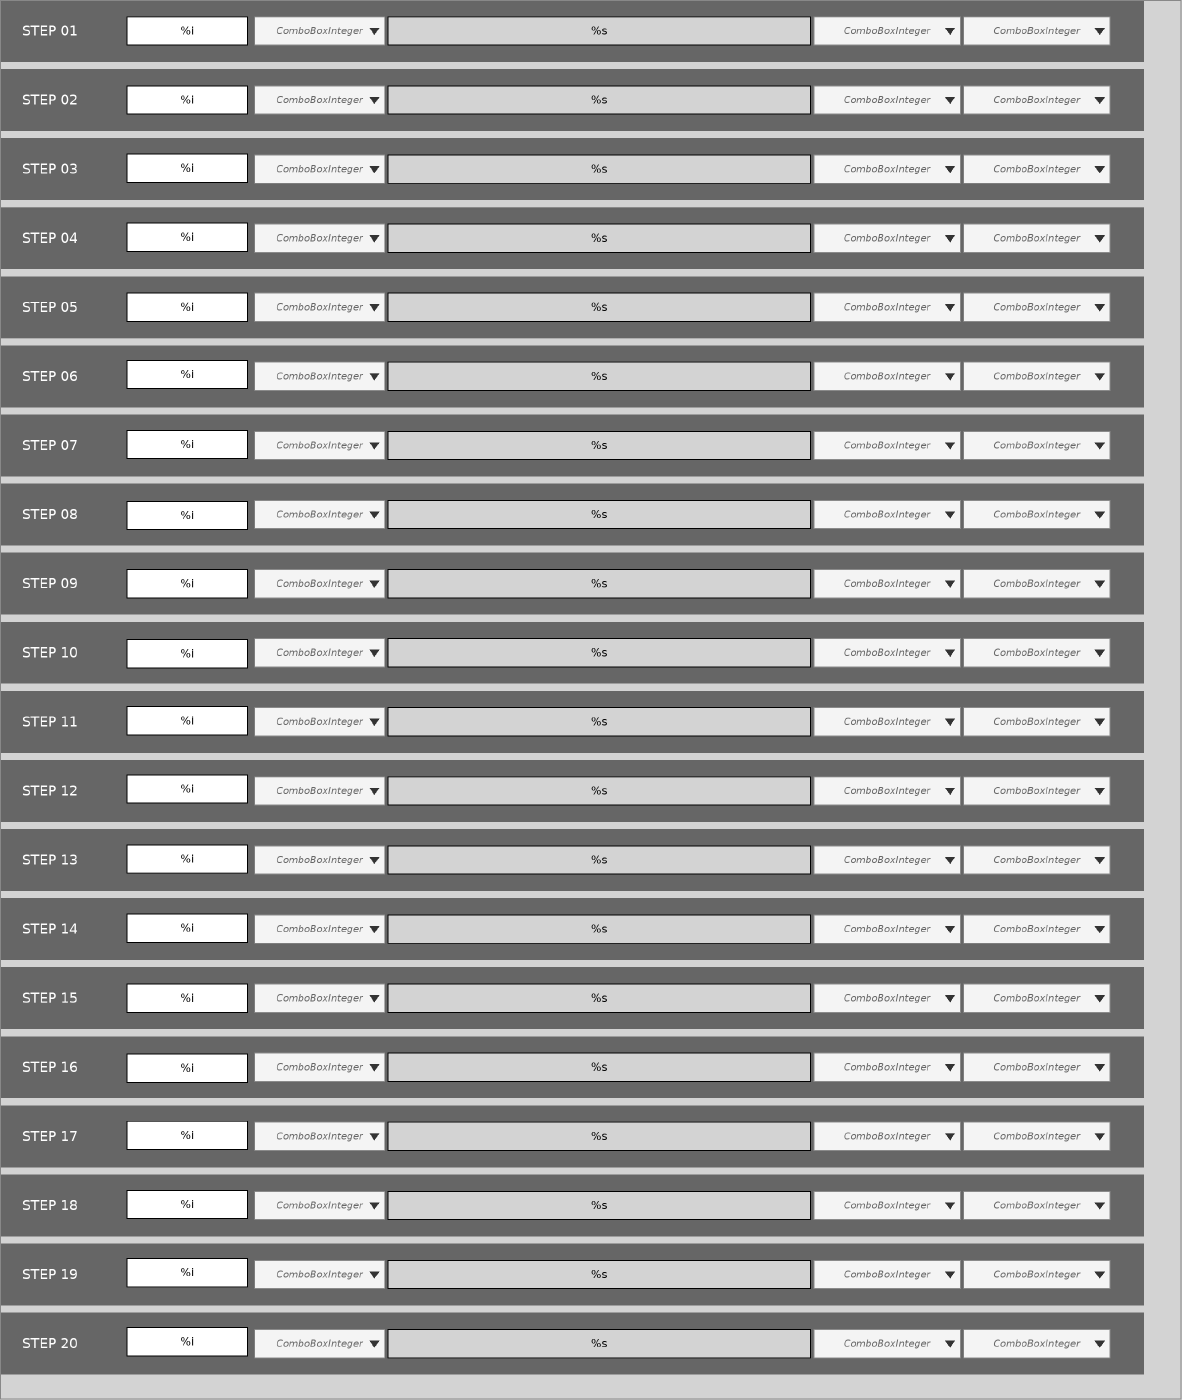
VISUALIZATION Popup_RecipeConfiguration  // 1232x1459
    RoundedRectangle (9,6 107x50)
    Rectangle (0,0 1232x1459)
    RoundedRectangle (0,360 1192x64)
    Label (20,380 103x24), "STEP 06"
    ComboBoxInteger (265,377 136x30), variable: Global_Variables_Arm_Persistent.DSA1fbPnpSequenceMemoryStore.DsA1inPnpSequenceMemory.ARiStnSeqRepNo[6], text list: 'RecipeNo'
    RoundedRectangle (404,377 441x30), "%s", text variable: Global_Variables_HMI_Function.sRecipeDescriptionStep[6]
    ComboBoxInteger (848,377 153x30), variable: Global_Variables_Arm_Persistent.DSA1fbPnpSequenceMemoryStore.DsA1inPnpSequenceMemory.ARiUpPickPatternNo[6], text list: 'TextList_1_20_Speed'
    ComboBoxInteger (1004,377 153x30), variable: Global_Variables_Arm_Persistent.DSA1fbPnpSequenceMemoryStore.DsA1inPnpSequenceMemory.ARiDownTransferPatternNo[6], text list: 'TextList_1_20_Speed'
    RoundedRectangle (0,432 1192x64)
    Label (20,452 103x24), "STEP 07"
    ComboBoxInteger (265,449 136x30), variable: Global_Variables_Arm_Persistent.DSA1fbPnpSequenceMemoryStore.DsA1inPnpSequenceMemory.ARiStnSeqRepNo[7], text list: 'RecipeNo'
    RoundedRectangle (404,449 441x30), "%s", text variable: Global_Variables_HMI_Function.sRecipeDescriptionStep[7]
    ComboBoxInteger (848,449 153x30), variable: Global_Variables_Arm_Persistent.DSA1fbPnpSequenceMemoryStore.DsA1inPnpSequenceMemory.ARiUpPickPatternNo[7], text list: 'TextList_1_20_Speed'
    ComboBoxInteger (1004,449 153x30), variable: Global_Variables_Arm_Persistent.DSA1fbPnpSequenceMemoryStore.DsA1inPnpSequenceMemory.ARiDownTransferPatternNo[7], text list: 'TextList_1_20_Speed'
    RoundedRectangle (0,504 1192x64)
    Label (20,524 103x24), "STEP 08"
    ComboBoxInteger (265,521 136x30), variable: Global_Variables_Arm_Persistent.DSA1fbPnpSequenceMemoryStore.DsA1inPnpSequenceMemory.ARiStnSeqRepNo[8], text list: 'RecipeNo'
    RoundedRectangle (404,521 441x30), "%s", text variable: Global_Variables_HMI_Function.sRecipeDescriptionStep[8]
    ComboBoxInteger (848,521 153x30), variable: Global_Variables_Arm_Persistent.DSA1fbPnpSequenceMemoryStore.DsA1inPnpSequenceMemory.ARiUpPickPatternNo[8], text list: 'TextList_1_20_Speed'
    ComboBoxInteger (1004,521 153x30), variable: Global_Variables_Arm_Persistent.DSA1fbPnpSequenceMemoryStore.DsA1inPnpSequenceMemory.ARiDownTransferPatternNo[8], text list: 'TextList_1_20_Speed'
    RoundedRectangle (0,576 1192x64)
    Label (20,596 103x24), "STEP 09"
    ComboBoxInteger (265,593 136x30), variable: Global_Variables_Arm_Persistent.DSA1fbPnpSequenceMemoryStore.DsA1inPnpSequenceMemory.ARiStnSeqRepNo[9], text list: 'RecipeNo'
    RoundedRectangle (404,593 441x30), "%s", text variable: Global_Variables_HMI_Function.sRecipeDescriptionStep[9]
    ComboBoxInteger (848,593 153x30), variable: Global_Variables_Arm_Persistent.DSA1fbPnpSequenceMemoryStore.DsA1inPnpSequenceMemory.ARiUpPickPatternNo[9], text list: 'TextList_1_20_Speed'
    ComboBoxInteger (1004,593 153x30), variable: Global_Variables_Arm_Persistent.DSA1fbPnpSequenceMemoryStore.DsA1inPnpSequenceMemory.ARiDownTransferPatternNo[9], text list: 'TextList_1_20_Speed'
    RoundedRectangle (0,648 1192x64)
    Label (20,668 103x24), "STEP 10"
    ComboBoxInteger (265,665 136x30), variable: Global_Variables_Arm_Persistent.DSA1fbPnpSequenceMemoryStore.DsA1inPnpSequenceMemory.ARiStnSeqRepNo[10], text list: 'RecipeNo'
    RoundedRectangle (404,665 441x30), "%s", text variable: Global_Variables_HMI_Function.sRecipeDescriptionStep[10]
    ComboBoxInteger (848,665 153x30), variable: Global_Variables_Arm_Persistent.DSA1fbPnpSequenceMemoryStore.DsA1inPnpSequenceMemory.ARiUpPickPatternNo[10], text list: 'TextList_1_20_Speed'
    ComboBoxInteger (1004,665 153x30), variable: Global_Variables_Arm_Persistent.DSA1fbPnpSequenceMemoryStore.DsA1inPnpSequenceMemory.ARiDownTransferPatternNo[10], text list: 'TextList_1_20_Speed'
    RoundedRectangle (0,0 1192x64)
    Label (20,20 103x24), "STEP 01"
    ComboBoxInteger (265,17 136x30), variable: Global_Variables_Arm_Persistent.DSA1fbPnpSequenceMemoryStore.DsA1inPnpSequenceMemory.ARiStnSeqRepNo[1], text list: 'RecipeNo'
    RoundedRectangle (404,17 441x30), "%s", text variable: Global_Variables_HMI_Function.sRecipeDescriptionStep[1]
    ComboBoxInteger (848,17 153x30), variable: Global_Variables_Arm_Persistent.DSA1fbPnpSequenceMemoryStore.DsA1inPnpSequenceMemory.ARiUpPickPatternNo[1], text list: 'TextList_1_20_Speed'
    ComboBoxInteger (1004,17 153x30), variable: Global_Variables_Arm_Persistent.DSA1fbPnpSequenceMemoryStore.DsA1inPnpSequenceMemory.ARiDownTransferPatternNo[1], text list: 'TextList_1_20_Speed'
    RoundedRectangle (0,72 1192x64)
    Label (20,92 103x24), "STEP 02"
    ComboBoxInteger (265,89 136x30), variable: Global_Variables_Arm_Persistent.DSA1fbPnpSequenceMemoryStore.DsA1inPnpSequenceMemory.ARiStnSeqRepNo[2], text list: 'RecipeNo'
    RoundedRectangle (404,89 441x30), "%s", text variable: Global_Variables_HMI_Function.sRecipeDescriptionStep[2]
    ComboBoxInteger (848,89 153x30), variable: Global_Variables_Arm_Persistent.DSA1fbPnpSequenceMemoryStore.DsA1inPnpSequenceMemory.ARiUpPickPatternNo[2], text list: 'TextList_1_20_Speed'
        p1601986498: ''
    ComboBoxInteger (1004,89 153x30), variable: Global_Variables_Arm_Persistent.DSA1fbPnpSequenceMemoryStore.DsA1inPnpSequenceMemory.ARiDownTransferPatternNo[2], text list: 'TextList_1_20_Speed'
    RoundedRectangle (0,144 1192x64)
    Label (20,164 103x24), "STEP 03"
    ComboBoxInteger (265,161 136x30), variable: Global_Variables_Arm_Persistent.DSA1fbPnpSequenceMemoryStore.DsA1inPnpSequenceMemory.ARiStnSeqRepNo[3], text list: 'RecipeNo'
    RoundedRectangle (404,161 441x30), "%s", text variable: Global_Variables_HMI_Function.sRecipeDescriptionStep[3]
    ComboBoxInteger (1004,161 153x30), variable: Global_Variables_Arm_Persistent.DSA1fbPnpSequenceMemoryStore.DsA1inPnpSequenceMemory.ARiDownTransferPatternNo[3], text list: 'TextList_1_20_Speed'
    RoundedRectangle (0,216 1192x64)
    Label (20,236 103x24), "STEP 04"
    ComboBoxInteger (265,233 136x30), variable: Global_Variables_Arm_Persistent.DSA1fbPnpSequenceMemoryStore.DsA1inPnpSequenceMemory.ARiStnSeqRepNo[4], text list: 'RecipeNo'
    RoundedRectangle (404,233 441x30), "%s", text variable: Global_Variables_HMI_Function.sRecipeDescriptionStep[4]
    ComboBoxInteger (848,233 153x30), variable: Global_Variables_Arm_Persistent.DSA1fbPnpSequenceMemoryStore.DsA1inPnpSequenceMemory.ARiUpPickPatternNo[4], text list: 'TextList_1_20_Speed'
    ComboBoxInteger (1004,233 153x30), variable: Global_Variables_Arm_Persistent.DSA1fbPnpSequenceMemoryStore.DsA1inPnpSequenceMemory.ARiDownTransferPatternNo[4], text list: 'TextList_1_20_Speed'
    RoundedRectangle (0,288 1192x64)
    Label (20,308 103x24), "STEP 05"
    ComboBoxInteger (265,305 136x30), variable: Global_Variables_Arm_Persistent.DSA1fbPnpSequenceMemoryStore.DsA1inPnpSequenceMemory.ARiStnSeqRepNo[5], text list: 'RecipeNo'
    RoundedRectangle (404,305 441x30), "%s", text variable: Global_Variables_HMI_Function.sRecipeDescriptionStep[5]
    ComboBoxInteger (848,305 153x30), variable: Global_Variables_Arm_Persistent.DSA1fbPnpSequenceMemoryStore.DsA1inPnpSequenceMemory.ARiUpPickPatternNo[5], text list: 'TextList_1_20_Speed'
    ComboBoxInteger (1004,305 153x30), variable: Global_Variables_Arm_Persistent.DSA1fbPnpSequenceMemoryStore.DsA1inPnpSequenceMemory.ARiDownTransferPatternNo[5], text list: 'TextList_1_20_Speed'
    RoundedRectangle (0,1080 1192x64)
    Label (20,1100 103x24), "STEP 16"
    ComboBoxInteger (265,1097 136x30), variable: Global_Variables_Arm_Persistent.DSA1fbPnpSequenceMemoryStore.DsA1inPnpSequenceMemory.ARiStnSeqRepNo[16], text list: 'RecipeNo'
    RoundedRectangle (404,1097 441x30), "%s", text variable: Global_Variables_HMI_Function.sRecipeDescriptionStep[16]
    ComboBoxInteger (848,1097 153x30), variable: Global_Variables_Arm_Persistent.DSA1fbPnpSequenceMemoryStore.DsA1inPnpSequenceMemory.ARiUpPickPatternNo[16], text list: 'TextList_1_20_Speed'
    ComboBoxInteger (1004,1097 153x30), variable: Global_Variables_Arm_Persistent.DSA1fbPnpSequenceMemoryStore.DsA1inPnpSequenceMemory.ARiDownTransferPatternNo[16], text list: 'TextList_1_20_Speed'
    RoundedRectangle (0,1152 1192x64)
    Label (20,1172 103x24), "STEP 17"
    ComboBoxInteger (265,1169 136x30), variable: Global_Variables_Arm_Persistent.DSA1fbPnpSequenceMemoryStore.DsA1inPnpSequenceMemory.ARiStnSeqRepNo[17], text list: 'RecipeNo'
    RoundedRectangle (404,1169 441x30), "%s", text variable: Global_Variables_HMI_Function.sRecipeDescriptionStep[17]
    ComboBoxInteger (848,1169 153x30), variable: Global_Variables_Arm_Persistent.DSA1fbPnpSequenceMemoryStore.DsA1inPnpSequenceMemory.ARiUpPickPatternNo[17], text list: 'TextList_1_20_Speed'
    ComboBoxInteger (1004,1169 153x30), variable: Global_Variables_Arm_Persistent.DSA1fbPnpSequenceMemoryStore.DsA1inPnpSequenceMemory.ARiDownTransferPatternNo[17], text list: 'TextList_1_20_Speed'
    RoundedRectangle (0,1224 1192x64)
    Label (20,1244 103x24), "STEP 18"
    ComboBoxInteger (265,1241 136x30), variable: Global_Variables_Arm_Persistent.DSA1fbPnpSequenceMemoryStore.DsA1inPnpSequenceMemory.ARiStnSeqRepNo[18], text list: 'RecipeNo'
    RoundedRectangle (404,1241 441x30), "%s", text variable: Global_Variables_HMI_Function.sRecipeDescriptionStep[18]
    ComboBoxInteger (848,1241 153x30), variable: Global_Variables_Arm_Persistent.DSA1fbPnpSequenceMemoryStore.DsA1inPnpSequenceMemory.ARiUpPickPatternNo[18], text list: 'TextList_1_20_Speed'
    ComboBoxInteger (1004,1241 153x30), variable: Global_Variables_Arm_Persistent.DSA1fbPnpSequenceMemoryStore.DsA1inPnpSequenceMemory.ARiDownTransferPatternNo[18], text list: 'TextList_1_20_Speed'
    RoundedRectangle (0,1296 1192x64)
    Label (20,1316 103x24), "STEP 19"
    ComboBoxInteger (265,1313 136x30), variable: Global_Variables_Arm_Persistent.DSA1fbPnpSequenceMemoryStore.DsA1inPnpSequenceMemory.ARiStnSeqRepNo[19], text list: 'RecipeNo'
    RoundedRectangle (404,1313 441x30), "%s", text variable: Global_Variables_HMI_Function.sRecipeDescriptionStep[19]
    ComboBoxInteger (848,1313 153x30), variable: Global_Variables_Arm_Persistent.DSA1fbPnpSequenceMemoryStore.DsA1inPnpSequenceMemory.ARiUpPickPatternNo[19], text list: 'TextList_1_20_Speed'
        p1601986498: ''
    ComboBoxInteger (1004,1313 153x30), variable: Global_Variables_Arm_Persistent.DSA1fbPnpSequenceMemoryStore.DsA1inPnpSequenceMemory.ARiDownTransferPatternNo[19], text list: 'TextList_1_20_Speed'
    RoundedRectangle (0,1368 1192x64)
    Label (20,1388 103x24), "STEP 20"
    ComboBoxInteger (265,1385 136x30), variable: Global_Variables_Arm_Persistent.DSA1fbPnpSequenceMemoryStore.DsA1inPnpSequenceMemory.ARiStnSeqRepNo[20], text list: 'RecipeNo'
    RoundedRectangle (404,1385 441x30), "%s", text variable: Global_Variables_HMI_Function.sRecipeDescriptionStep[20]
    ComboBoxInteger (848,1385 153x30), variable: Global_Variables_Arm_Persistent.DSA1fbPnpSequenceMemoryStore.DsA1inPnpSequenceMemory.ARiUpPickPatternNo[20], text list: 'TextList_1_20_Speed'
    ComboBoxInteger (1004,1385 153x30), variable: Global_Variables_Arm_Persistent.DSA1fbPnpSequenceMemoryStore.DsA1inPnpSequenceMemory.ARiDownTransferPatternNo[20], text list: 'TextList_1_20_Speed'
    RoundedRectangle (0,720 1192x64)
    Label (20,740 103x24), "STEP 11"
    ComboBoxInteger (265,737 136x30), variable: Global_Variables_Arm_Persistent.DSA1fbPnpSequenceMemoryStore.DsA1inPnpSequenceMemory.ARiStnSeqRepNo[11], text list: 'RecipeNo'
    RoundedRectangle (404,737 441x30), "%s", text variable: Global_Variables_HMI_Function.sRecipeDescriptionStep[11]
    ComboBoxInteger (848,737 153x30), variable: Global_Variables_Arm_Persistent.DSA1fbPnpSequenceMemoryStore.DsA1inPnpSequenceMemory.ARiUpPickPatternNo[11], text list: 'TextList_1_20_Speed'
    ComboBoxInteger (1004,737 153x30), variable: Global_Variables_Arm_Persistent.DSA1fbPnpSequenceMemoryStore.DsA1inPnpSequenceMemory.ARiDownTransferPatternNo[11], text list: 'TextList_1_20_Speed'
    RoundedRectangle (0,792 1192x64)
    Label (20,812 103x24), "STEP 12"
    ComboBoxInteger (265,809 136x30), variable: Global_Variables_Arm_Persistent.DSA1fbPnpSequenceMemoryStore.DsA1inPnpSequenceMemory.ARiStnSeqRepNo[12], text list: 'RecipeNo'
    RoundedRectangle (404,809 441x30), "%s", text variable: Global_Variables_HMI_Function.sRecipeDescriptionStep[12]
    ComboBoxInteger (848,809 153x30), variable: Global_Variables_Arm_Persistent.DSA1fbPnpSequenceMemoryStore.DsA1inPnpSequenceMemory.ARiUpPickPatternNo[12], text list: 'TextList_1_20_Speed'
    ComboBoxInteger (1004,809 153x30), variable: Global_Variables_Arm_Persistent.DSA1fbPnpSequenceMemoryStore.DsA1inPnpSequenceMemory.ARiDownTransferPatternNo[12], text list: 'TextList_1_20_Speed'
    RoundedRectangle (0,864 1192x64)
    Label (20,884 103x24), "STEP 13"
    ComboBoxInteger (265,881 136x30), variable: Global_Variables_Arm_Persistent.DSA1fbPnpSequenceMemoryStore.DsA1inPnpSequenceMemory.ARiStnSeqRepNo[13], text list: 'RecipeNo'
    RoundedRectangle (404,881 441x30), "%s", text variable: Global_Variables_HMI_Function.sRecipeDescriptionStep[13]
    ComboBoxInteger (848,881 153x30), variable: Global_Variables_Arm_Persistent.DSA1fbPnpSequenceMemoryStore.DsA1inPnpSequenceMemory.ARiUpPickPatternNo[13], text list: 'TextList_1_20_Speed'
    ComboBoxInteger (1004,881 153x30), variable: Global_Variables_Arm_Persistent.DSA1fbPnpSequenceMemoryStore.DsA1inPnpSequenceMemory.ARiDownTransferPatternNo[13], text list: 'TextList_1_20_Speed'
    RoundedRectangle (0,936 1192x64)
    Label (20,956 103x24), "STEP 14"
    ComboBoxInteger (265,953 136x30), variable: Global_Variables_Arm_Persistent.DSA1fbPnpSequenceMemoryStore.DsA1inPnpSequenceMemory.ARiStnSeqRepNo[14], text list: 'RecipeNo'
    RoundedRectangle (404,953 441x30), "%s", text variable: Global_Variables_HMI_Function.sRecipeDescriptionStep[14]
    ComboBoxInteger (848,953 153x30), variable: Global_Variables_Arm_Persistent.DSA1fbPnpSequenceMemoryStore.DsA1inPnpSequenceMemory.ARiUpPickPatternNo[14], text list: 'TextList_1_20_Speed'
    ComboBoxInteger (1004,953 153x30), variable: Global_Variables_Arm_Persistent.DSA1fbPnpSequenceMemoryStore.DsA1inPnpSequenceMemory.ARiDownTransferPatternNo[14], text list: 'TextList_1_20_Speed'
    RoundedRectangle (0,1008 1192x64)
    Label (20,1028 103x24), "STEP 15"
    ComboBoxInteger (265,1025 136x30), variable: Global_Variables_Arm_Persistent.DSA1fbPnpSequenceMemoryStore.DsA1inPnpSequenceMemory.ARiStnSeqRepNo[15], text list: 'RecipeNo'
    RoundedRectangle (404,1025 441x30), "%s", text variable: Global_Variables_HMI_Function.sRecipeDescriptionStep[15]
    ComboBoxInteger (848,1025 153x30), variable: Global_Variables_Arm_Persistent.DSA1fbPnpSequenceMemoryStore.DsA1inPnpSequenceMemory.ARiUpPickPatternNo[15], text list: 'TextList_1_20_Speed'
    ComboBoxInteger (1004,1025 153x30), variable: Global_Variables_Arm_Persistent.DSA1fbPnpSequenceMemoryStore.DsA1inPnpSequenceMemory.ARiDownTransferPatternNo[15], text list: 'TextList_1_20_Speed'
    ComboBoxInteger (848,161 153x30), variable: Global_Variables_Arm_Persistent.DSA1fbPnpSequenceMemoryStore.DsA1inPnpSequenceMemory.ARiUpPickPatternNo[3], text list: 'TextList_1_20_Speed'
    RoundedRectangle (132,17 126x30), "%i", text variable: Global_Variables_Arm_Persistent.DSA1fbPnpSequenceMemoryStore.DsA1inPnpSequenceMemory.ARiTransferStationNo[1]
        OnMouseDown: write the text variable via VisuDialogs.Numpad
    RoundedRectangle (132,89 126x30), "%i", text variable: Global_Variables_Arm_Persistent.DSA1fbPnpSequenceMemoryStore.DsA1inPnpSequenceMemory.ARiTransferStationNo[2]
        OnMouseDown: write the text variable via VisuDialogs.Numpad
    RoundedRectangle (132,160 126x30), "%i", text variable: Global_Variables_Arm_Persistent.DSA1fbPnpSequenceMemoryStore.DsA1inPnpSequenceMemory.ARiTransferStationNo[3]
        OnMouseDown: write the text variable via VisuDialogs.Numpad
    RoundedRectangle (132,232 126x30), "%i", text variable: Global_Variables_Arm_Persistent.DSA1fbPnpSequenceMemoryStore.DsA1inPnpSequenceMemory.ARiTransferStationNo[4]
        OnMouseDown: write the text variable via VisuDialogs.Numpad
    RoundedRectangle (132,305 126x30), "%i", text variable: Global_Variables_Arm_Persistent.DSA1fbPnpSequenceMemoryStore.DsA1inPnpSequenceMemory.ARiTransferStationNo[5]
        OnMouseDown: write the text variable via VisuDialogs.Numpad
    RoundedRectangle (132,375 126x30), "%i", text variable: Global_Variables_Arm_Persistent.DSA1fbPnpSequenceMemoryStore.DsA1inPnpSequenceMemory.ARiTransferStationNo[6]
        OnMouseDown: write the text variable via VisuDialogs.Numpad
    RoundedRectangle (132,448 126x30), "%i", text variable: Global_Variables_Arm_Persistent.DSA1fbPnpSequenceMemoryStore.DsA1inPnpSequenceMemory.ARiTransferStationNo[7]
        OnMouseDown: write the text variable via VisuDialogs.Numpad
    RoundedRectangle (132,522 126x30), "%i", text variable: Global_Variables_Arm_Persistent.DSA1fbPnpSequenceMemoryStore.DsA1inPnpSequenceMemory.ARiTransferStationNo[8]
        OnMouseDown: write the text variable via VisuDialogs.Numpad
    RoundedRectangle (132,593 126x30), "%i", text variable: Global_Variables_Arm_Persistent.DSA1fbPnpSequenceMemoryStore.DsA1inPnpSequenceMemory.ARiTransferStationNo[9]
        OnMouseDown: write the text variable via VisuDialogs.Numpad
    RoundedRectangle (132,666 126x30), "%i", text variable: Global_Variables_Arm_Persistent.DSA1fbPnpSequenceMemoryStore.DsA1inPnpSequenceMemory.ARiTransferStationNo[10]
        OnMouseDown: write the text variable via VisuDialogs.Numpad
    RoundedRectangle (132,736 126x30), "%i", text variable: Global_Variables_Arm_Persistent.DSA1fbPnpSequenceMemoryStore.DsA1inPnpSequenceMemory.ARiTransferStationNo[11]
        OnMouseDown: write the text variable via VisuDialogs.Numpad
    RoundedRectangle (132,807 126x30), "%i", text variable: Global_Variables_Arm_Persistent.DSA1fbPnpSequenceMemoryStore.DsA1inPnpSequenceMemory.ARiTransferStationNo[12]
        OnMouseDown: write the text variable via VisuDialogs.Numpad
    RoundedRectangle (132,880 126x30), "%i", text variable: Global_Variables_Arm_Persistent.DSA1fbPnpSequenceMemoryStore.DsA1inPnpSequenceMemory.ARiTransferStationNo[13]
        OnMouseDown: write the text variable via VisuDialogs.Numpad
    RoundedRectangle (132,952 126x30), "%i", text variable: Global_Variables_Arm_Persistent.DSA1fbPnpSequenceMemoryStore.DsA1inPnpSequenceMemory.ARiTransferStationNo[14]
        OnMouseDown: write the text variable via VisuDialogs.Numpad
    RoundedRectangle (132,1025 126x30), "%i", text variable: Global_Variables_Arm_Persistent.DSA1fbPnpSequenceMemoryStore.DsA1inPnpSequenceMemory.ARiTransferStationNo[15]
        OnMouseDown: write the text variable via VisuDialogs.Numpad
    RoundedRectangle (132,1098 126x30), "%i", text variable: Global_Variables_Arm_Persistent.DSA1fbPnpSequenceMemoryStore.DsA1inPnpSequenceMemory.ARiTransferStationNo[16]
        OnMouseDown: write the text variable via VisuDialogs.Numpad
    RoundedRectangle (132,1168 126x30), "%i", text variable: Global_Variables_Arm_Persistent.DSA1fbPnpSequenceMemoryStore.DsA1inPnpSequenceMemory.ARiTransferStationNo[17]
        OnMouseDown: write the text variable via VisuDialogs.Numpad
    RoundedRectangle (132,1240 126x30), "%i", text variable: Global_Variables_Arm_Persistent.DSA1fbPnpSequenceMemoryStore.DsA1inPnpSequenceMemory.ARiTransferStationNo[18]
        OnMouseDown: write the text variable via VisuDialogs.Numpad
    RoundedRectangle (132,1311 126x30), "%i", text variable: Global_Variables_Arm_Persistent.DSA1fbPnpSequenceMemoryStore.DsA1inPnpSequenceMemory.ARiTransferStationNo[19]
        OnMouseDown: write the text variable via VisuDialogs.Numpad
    RoundedRectangle (132,1383 126x30), "%i", text variable: Global_Variables_Arm_Persistent.DSA1fbPnpSequenceMemoryStore.DsA1inPnpSequenceMemory.ARiTransferStationNo[20]
        OnMouseDown: write the text variable via VisuDialogs.Numpad
END_VISUALIZATION

(* stored: Version 1.1.0.1, ProductVersion 3.1.4024.12
   Visu Popup_RecipeConfiguration: Id {8f3979a9-9c0a-42d7-8acb-abd8c0f2728d} *)
